FUNCTION_BLOCK ATM_AX_PULSE_RETRIG (* Standard timer function block (pulse) - retriggerable version *)
  (* Standard: 61499-2; Description: Copyright (c) 2023 HR Agrartechnik GmbH This program and the accompanying materials are made available under the terms of the Eclipse Public License 2.0 which is available at https://www.eclipse.org/legal/epl-2.0/ SPDX-License-Identifier: EPL-2.0 AT_AX_PULSE_RETRIG -- Impulse forming FB with AX/AT adapter interface (Retriggerable) The adapter input PT provides the pulse time (D1->PT). Generate an Impulse with a given Time. This FB makes an Impulse of Duration PT on the Output Q. New REQ restarts the timer. *)
  (* Version 1.0, 2026-04-19, Franz Höpfinger, HR Agrartechnik GmbH, retriggerable version *)
  PACKAGE adapter::events::unidirectional::timers;
  IMPORT eclipse4diac::core::TypeHash;
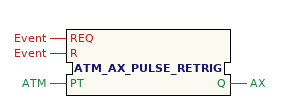
  EVENT_INPUT
    REQ; (* Service Request (Restarts the timer) *)
    R; (* Reset *)
  END_EVENT
  SOCKETS
    PT : adapter::types::unidirectional::ATM; (* Pulse time (AT adapter) *)
  END_SOCKETS
  PLUGS
    Q : adapter::types::unidirectional::AX; (* Timer output (AX adapter) *)
  END_PLUGS
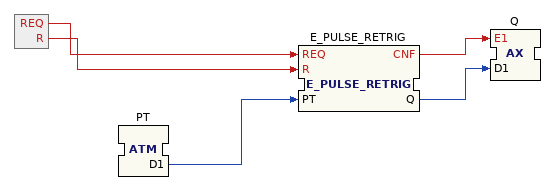
  FBS
    E_PULSE_RETRIG : iec61499::events::timers::E_PULSE_RETRIG;
  END_FBS
  EVENT_CONNECTIONS
    E_PULSE_RETRIG.CNF TO Q.E1;
    REQ TO E_PULSE_RETRIG.REQ;
    R TO E_PULSE_RETRIG.R;
  END_CONNECTIONS
  DATA_CONNECTIONS
    E_PULSE_RETRIG.Q TO Q.D1;
    PT.D1 TO E_PULSE_RETRIG.PT;
  END_CONNECTIONS
END_FUNCTION_BLOCK
